PROGRAM ControlFBD
VAR
	qxLampStarted	AT %Q* : BOOL;
	gxSliderAout 	AT %Q* : BOOL; 
	gxSliderAin 	AT %Q* : BOOL; 
	gxSliderBout 	AT %Q* : BOOL; 
	gxSliderBin 	AT %Q* : BOOL; 
	gxDrillDown 	AT %Q* : BOOL;
	gxDrillUp		AT %Q* : BOOL;
	
	ixButtonStart	AT %I* : BOOL;
	ixButtonStop	AT %I* : BOOL;
	ixSliderAout	AT %I* : BOOL;
	ixSliderAin		AT %I* : BOOL;
	ixSliderBout	AT %I* : BOOL;
	ixSliderBin		AT %I* : BOOL;
	ixDrillUp		AT %I* : BOOL;
	ixDrillDown		AT %I* : BOOL;

	drilled: BOOL;
	new_start: BOOL;
END_VAR

VAR_INPUT
	mxSlideBin: BOOL;
END_VAR

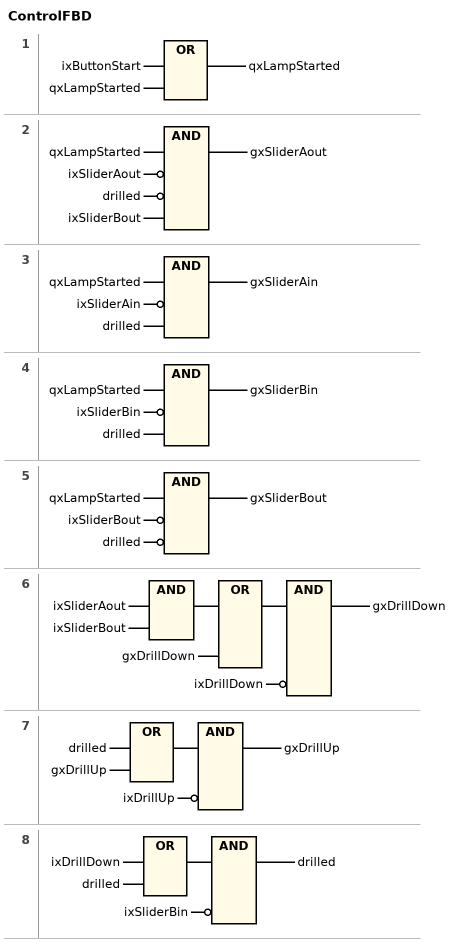
// NETWORK 1
qxLampStarted := ixButtonStart OR qxLampStarted;

// NETWORK 2
gxSliderAout := qxLampStarted AND NOT ixSliderAout AND NOT drilled AND ixSliderBout;

// NETWORK 3
gxSliderAin := qxLampStarted AND NOT ixSliderAin AND drilled;

// NETWORK 4
gxSliderBin := qxLampStarted AND NOT ixSliderBin AND drilled;

// NETWORK 5
gxSliderBout := qxLampStarted AND NOT ixSliderBout AND NOT drilled;

// NETWORK 6
gxDrillDown := (ixSliderAout AND ixSliderBout OR gxDrillDown) AND NOT ixDrillDown;

// NETWORK 7
gxDrillUp := (drilled OR gxDrillUp) AND NOT ixDrillUp;

// NETWORK 8
drilled := (ixDrillDown OR drilled) AND NOT ixSliderBin;

END_PROGRAM

(* stored: Version 1.1.0.1, ProductVersion 3.1.4024.9
   POU ControlFBD: Id {441bf843-2f16-42db-a10b-d561aec11b1f}, SpecialFunc None *)
